// TIA Portal V20 export
TYPE "LER_typeEmRelation"
// stored: Access Published
   STRUCT
      "Bool" { ExternalWritable := 'False'} : Array[0..99] of Bool;   // User Define
      LReal { ExternalWritable := 'False'} : Array[0..19] of LReal;   // User Define
      softCam { ExternalWritable := 'False'} : Array[0..15] of "LER_typeSoftCamRelation";   // Axis Position Check
      cmStatus { ExternalWritable := 'False'} : "LER_typeCmStatus";   // Control Modules Status
      sequence { ExternalWritable := 'False'} : Array[0..19] of "LER_typeSequenceRelation";   // Em Sequence
   END_STRUCT;
END_TYPE
